Staubli VAL3: init.pgx

public program init()
begin

  // Do nothing
  // See start() program for more details

end
